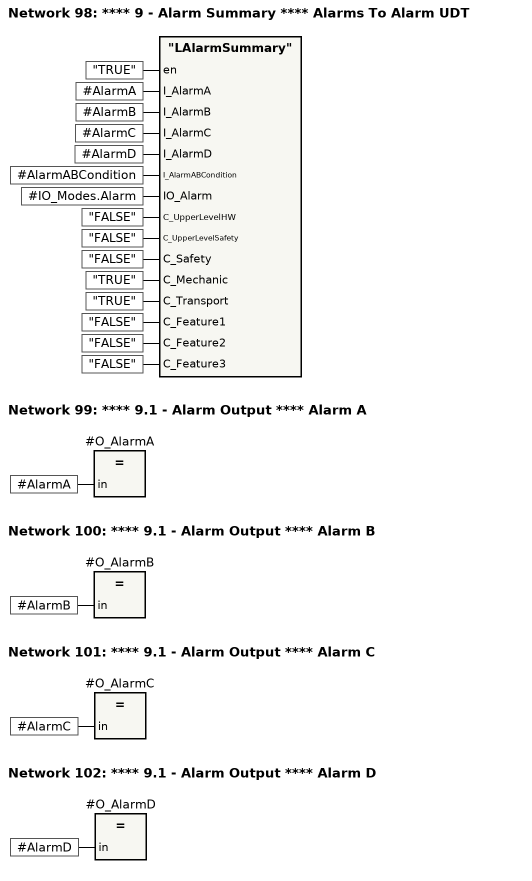
   IF "TRUE" THEN
       "LAlarmSummary"(I_AlarmA := #AlarmA,
                       I_AlarmB := #AlarmB,
                       I_AlarmC := #AlarmC,
                       I_AlarmD := #AlarmD,
                       I_AlarmABCondition := #AlarmABCondition,
                       IO_Alarm := #IO_Modes.Alarm,
                       C_UpperLevelHW := "FALSE",
                       C_UpperLevelSafety := "FALSE",
                       C_Safety := "FALSE",
                       C_Mechanic := "TRUE",
                       C_Transport := "TRUE",
                       C_Feature1 := "FALSE",
                       C_Feature2 := "FALSE",
                       C_Feature3 := "FALSE");
   END_IF;
END_REGION

REGION Network 99: **** 9.1 - Alarm Output **** Alarm A
   // Alarm A
   #O_AlarmA := #AlarmA;
END_REGION

REGION Network 100: **** 9.1 - Alarm Output **** Alarm B
   // Alarm B
   #O_AlarmB := #AlarmB;
END_REGION

REGION Network 101: **** 9.1 - Alarm Output **** Alarm C
   // Alarm C
   #O_AlarmC := #AlarmC;
END_REGION

REGION Network 102: **** 9.1 - Alarm Output **** Alarm D
   // Alarm D
   #O_AlarmD := #AlarmD;
END_REGION

REGION Network 103: **** 9.2 - Alarm DWord**** Alarm To DWord
   // Alarm To Word
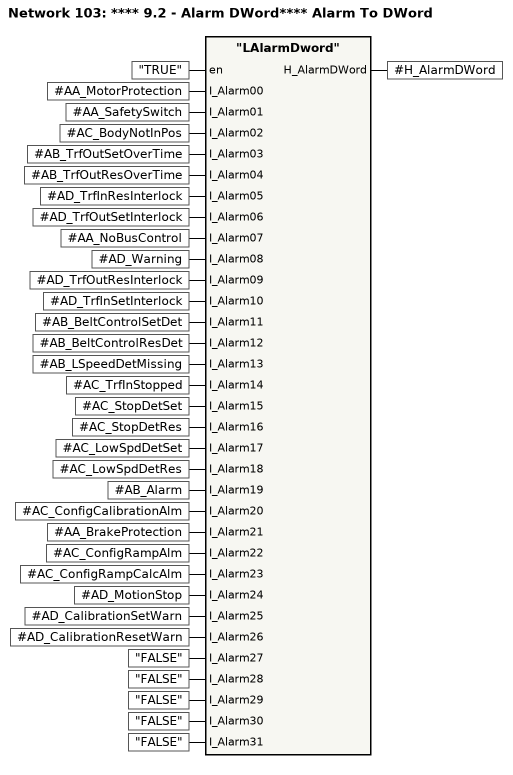
   IF "TRUE" THEN
       "LAlarmDword"(I_Alarm00 := #AA_MotorProtection,
                     I_Alarm01 := #AA_SafetySwitch,
                     I_Alarm02 := #AC_BodyNotInPos,
                     I_Alarm03 := #AB_TrfOutSetOverTime,
                     I_Alarm04 := #AB_TrfOutResOverTime,
                     I_Alarm05 := #AD_TrfInResInterlock,
                     I_Alarm06 := #AD_TrfOutSetInterlock,
                     I_Alarm07 := #AA_NoBusControl,
                     I_Alarm08 := #AD_Warning,
                     I_Alarm09 := #AD_TrfOutResInterlock,
                     I_Alarm10 := #AD_TrfInSetInterlock,
                     I_Alarm11 := #AB_BeltControlSetDet,
                     I_Alarm12 := #AB_BeltControlResDet,
                     I_Alarm13 := #AB_LSpeedDetMissing,
                     I_Alarm14 := #AC_TrfInStopped,
                     I_Alarm15 := #AC_StopDetSet,
                     I_Alarm16 := #AC_StopDetRes,
                     I_Alarm17 := #AC_LowSpdDetSet,
                     I_Alarm18 := #AC_LowSpdDetRes,
                     I_Alarm19 := #AB_Alarm,
                     I_Alarm20 := #AC_ConfigCalibrationAlm,
                     I_Alarm21 := #AA_BrakeProtection,
                     I_Alarm22 := #AC_ConfigRampAlm,
                     I_Alarm23 := #AC_ConfigRampCalcAlm,
                     I_Alarm24 := #AD_MotionStop,
                     I_Alarm25 := #AD_CalibrationSetWarn,
                     I_Alarm26 := #AD_CalibrationResetWarn,
                     I_Alarm27 := "FALSE",
                     I_Alarm28 := "FALSE",
                     I_Alarm29 := "FALSE",
                     I_Alarm30 := "FALSE",
                     I_Alarm31 := "FALSE",
                     H_AlarmDWord => #H_AlarmDWord);
   END_IF;
END_REGION
END_FUNCTION_BLOCK
